VAR
    fbCourseControl : FB_CourseDifferenceControl;
END_VAR

// 调用航向差控制功能块
fbCourseControl(
    KOMPASS_GRAD := g_KOMPASS_GRAD,
    KURS := g_KURS,
    KURS_DIFF := g_KURS_DIFF,
    ErrorFlag := g_ErrorFlag,
    ErrorCode := g_ErrorCode
);

(* stored: Name MAIN, Version 1.0.0.1, ProductVersion 3.1.4024.17
   POU: Type Program *)
